TYPE ST_Filter :
STRUCT
	fSignal 			: LREAL;
	fFilteredSignal 	: LREAL;
	fDanielFilter		: LREAL;
	fDanielFilter2		: LREAL;
END_STRUCT
END_TYPE

(* stored: Version 1.1.0.1
   DUT ST_Filter: Id {ca5d853b-e0f0-4622-8ad3-3c591972b906} *)
